(* IEC 61131-3 sources: FishAndCat/factoryio/lesson2_st, 2 files *)

(* ---- belt_stop.st ---- *)
(* ============================================================
   belt_stop.st — 三课·第二课教具①:光电挡停传送带(10 行热身)
   目标:证明「CODESYS Control Win(软 PLC)→ OPC UA → Factory I/O」全链路通。
   Factory I/O 场景:From A to B(或任何“一条传送带+一个漫反射光电”的场景)。

   学生操作(亲手做,Codex 陪跑):
   1. CODESYS 新建标准工程(设备选 CODESYS Control Win V3 x64),POU 语言 ST;
   2. 把本文件的 VAR 段与逻辑段分别粘进 PLC_PRG 的声明区/实现区;
   3. 添加 Symbol Configuration(勾选 PLC_PRG 全部变量)→ 编译 → 下载 → RUN;
   4. Factory I/O:File→Drivers→OPC Client DA/UA→ 连本机 CODESYS,
      按下面注释把变量映射到场景部件(以 FIO 驱动窗口显示的实际 tag 为准);
   5. FIO 点 RUN(注意:FIO 的 RUN 和 CODESYS 的 RUN 是两个开关,都要开)。

   验收(教程口径):箱子走到光电前,传送带自动停;拿走箱子(FIO 里拖走
   或复位场景),按 Start 后带子再走。录 30 秒屏发回 Claude。
   ============================================================ *)
PROGRAM PLC_PRG
VAR
    // ---- 映射到 Factory I/O(名字→FIO 部件,方向以 PLC 视角) ----
    xSensor  : BOOL;    // ← FIO “Diffuse Sensor”(检测到箱子=TRUE)
    xStart   : BOOL;    // ← FIO “Start Button”(绿色,按下=TRUE)
    xStop    : BOOL;    // ← FIO “Stop Button”(红色,注意:FIO 惯例常闭,松开=TRUE、按下=FALSE)
    xBeltRun : BOOL;    // → FIO “Belt Conveyor”(TRUE=运转)
    // ---- 内部 ----
    xRun     : BOOL;    // 运行自保持
END_VAR

// 启停自保持:Start 置位;Stop(常闭断开)复位——工业启停最小骨架
IF xStart THEN
    xRun := TRUE;
END_IF
IF NOT xStop THEN                   // 常闭按钮:按下时信号变 FALSE
    xRun := FALSE;
END_IF

// 核心一行:运行中 且 光电没被挡住 → 带子转;箱子到位即停
xBeltRun := xRun AND NOT xSensor;
END_PROGRAM

(* 常见坑(卡住先看这里,再喊 Codex):
   1. 带子不转:FIO 是否 RUN?CODESYS 是否 RUN?两个开关缺一不可;
   2. 变量全灰/映射窗口空:Symbol Configuration 没下载——重新编译+下载;
   3. Stop 一按就永远停:你的场景 Stop 按钮可能是常开——把 NOT xStop 改成 xStop;
   4. 光电不变化:FIO 里传感器 tag 没映射到 xSensor,或映射了别的传感器。 *)

(* ---- crane_3boxes.st ---- *)
(* ============================================================
   crane_3boxes.st — 三课·第二课教具②:堆垛机按序入库 3 箱
   目标:用最小状态机把 3 个货箱依次送进 3 个不同格位——
        这是主线 ST(400 库位分配)在“带物理引擎的世界”里的微缩证据,
        录屏进决赛展望「孪生成熟度阶梯」L2 实证层。
   Factory I/O 场景:Automated Warehouse(内置 54 格)或 Stacker Crane 单元。

   接口约定(FIO Stacker Crane 部件,tag 名以 FIO 驱动窗口实际显示为准;
   若你的版本 tag 不同,只改变量映射,状态机骨架不动——对不上喊 Codex 陪查):
     → iTargetPos  写目标格位编号(FIO “Target Position”,1..54;0=入库口/原位)
     → xLift       叉臂动作(FIO “Lift”:TRUE=托起/放下动作,随场景定义)
     ← xMovingX    水平移动中(FIO “Moving X”)
     ← xMovingZ    垂直移动中(FIO “Moving Z”)
     ← xAtLoad     入库口有箱(光电/“Box at load”类传感器)
   学生操作流程同 belt_stop.st(粘贴→Symbol Configuration→下载→OPC 映射→双 RUN)。

   验收:按 Start 后,3 个箱子被依次放进格位 5 / 18 / 31(三个不同巷道位置,
   演示“算法指定格位”而不是“就近乱放”);全程无手动干预。录 30 秒屏。
   ============================================================ *)
PROGRAM PLC_PRG
VAR
    // ---- 映射到 Factory I/O ----
    xStart     : BOOL;                  // ← Start 按钮
    xAtLoad    : BOOL;                  // ← 入库口有箱传感器
    xMovingX   : BOOL;                  // ← 堆垛机水平移动中
    xMovingZ   : BOOL;                  // ← 堆垛机垂直移动中
    iTargetPos : INT;                   // → 目标格位(0=回入库口)
    xLift      : BOOL;                  // → 叉臂动作
    // ---- 内部 ----
    iStep      : INT := 0;              // 状态机:0待命 10取箱 20去目标 30放箱 40回程 90完成
    iBoxIdx    : INT := 0;              // 已入库箱数(0..3)
    aSlot      : ARRAY[1..3] OF INT := [5, 18, 31];   // “算法给定”的三个目标格位
    xBusy      : BOOL;                  // 堆垛机在动(两轴任一)
    tonSettle  : TON;                   // 到位去抖:停稳 0.5s 才算到位
    tonAlarm   : TON;                   // 单步看门狗:20s 不完成=报警(演示防呆)
    xStepAlarm : BOOL;
END_VAR

xBusy := xMovingX OR xMovingZ;
tonSettle(IN := NOT xBusy, PT := T#500MS);          // 停稳计时
tonAlarm(IN := (iStep > 0) AND (iStep < 90), PT := T#20S);
IF tonAlarm.Q THEN                                   // 看门狗:卡步报警并回待命
    xStepAlarm := TRUE;
    iStep := 0;
END_IF

CASE iStep OF
    0:  // 待命:按 Start 且入库口有箱 → 开始
        xLift := FALSE;
        iTargetPos := 0;                             // 停在入库口
        IF xStart AND xAtLoad AND (iBoxIdx < 3) THEN
            xStepAlarm := FALSE;
            iStep := 10;
        END_IF

    10: // 取箱:在入库口做叉取动作(FIO 里 Lift 在 load 位=取箱)
        xLift := TRUE;
        IF tonSettle.Q THEN                          // 动作到位(停稳)
            iStep := 20;
        END_IF

    20: // 载箱去目标格:写目标位,等两轴到位停稳
        iTargetPos := aSlot[iBoxIdx + 1];
        IF xBusy THEN
            iStep := 25;                             // 确认已起动,再等停稳(防“还没动就误判到位”)
        END_IF
    25:
        IF tonSettle.Q THEN
            iStep := 30;
        END_IF

    30: // 放箱:叉臂收回(FIO 里 Lift 复位=放下)
        xLift := FALSE;
        IF tonSettle.Q THEN
            iBoxIdx := iBoxIdx + 1;
            iStep := 40;
        END_IF

    40: // 空载回入库口,准备下一箱
        iTargetPos := 0;
        IF xBusy THEN
            iStep := 45;
        END_IF
    45:
        IF tonSettle.Q THEN
            IF iBoxIdx >= 3 THEN
                iStep := 90;                         // 3 箱完成
            ELSE
                iStep := 0;                          // 等下一箱(xAtLoad)
            END_IF
        END_IF

    90: // 完成:驻留(重跑=FIO 复位场景 + 这里手动把 iBoxIdx/iStep 清零)
        ;
END_CASE
END_PROGRAM

(* 教学点(Codex 讲评提纲,对应主线 ST 的同款手法):
   1. 状态机(CASE)= 主线 05_PRG_Main 同构:每步只做一件事,完成条件明确;
   2. “先确认起动、再等停稳”(20→25)= 防抖两段式,主线 fbAssign 的 xBusy/xDone 同思想;
   3. TON 看门狗 = 任何真实设备控制都要的防卡步兜底;
   4. aSlot 数组 = “格位由算法给”:第三课 3a 就是把这 3 个数换成评分函数算出来的。
   常见坑:堆垛机不动=Target Position 没映射或量纲不对(有的版本按格号、有的按毫米);
   Lift 语义相反=把 10/30 两步的 TRUE/FALSE 互换。 *)
